FUNCTION GetMinor : UINT
VAR_INPUT
END_VAR
VAR
END_VAR

GetMinor := Version.Minor;

END_FUNCTION

(* stored: Version 1.1.0.1, ProductVersion 3.1.4024.0
   POU GetMinor: Id {1fbace56-5b28-41f7-8956-22c86ea94342}, SpecialFunc None *)
